// TIA Portal V20 export
DATA_BLOCK "DB_ToteTracking"   // DB38
// stored: Access Published, MemoryReserve 100, Namespace Global
   VAR
      Conveyor : Array[_.gMinC1.._.gMaxC1] of "Global.TrackingData";
      Barcode : Array[_.gMinC1.._.gMaxC1] of String;
   END_VAR
BEGIN
END_DATA_BLOCK
